SUBAPPLICATION CONSTRUCT_DDS_TOPIC (* Construct DDS Topic *)
  (* Standard: 61499-2 *)
  (* Version 1.0, 2023-03-15, Tim Hesse *)
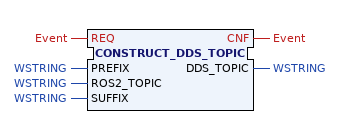
  EVENT_INPUT
    REQ; (* Normal Execution Request *)
  END_EVENT
  EVENT_OUTPUT
    CNF; (* Execution Confirmation *)
  END_EVENT
  VAR_INPUT
    PREFIX : WSTRING; (* Topic Prefix *)
    ROS2_TOPIC : WSTRING; (* ROS 2 Topic *)
    SUFFIX : WSTRING; (* Topic Suffix *)
  END_VAR
  VAR_OUTPUT
    DDS_TOPIC : WSTRING; (* DDS Topic *)
  END_VAR
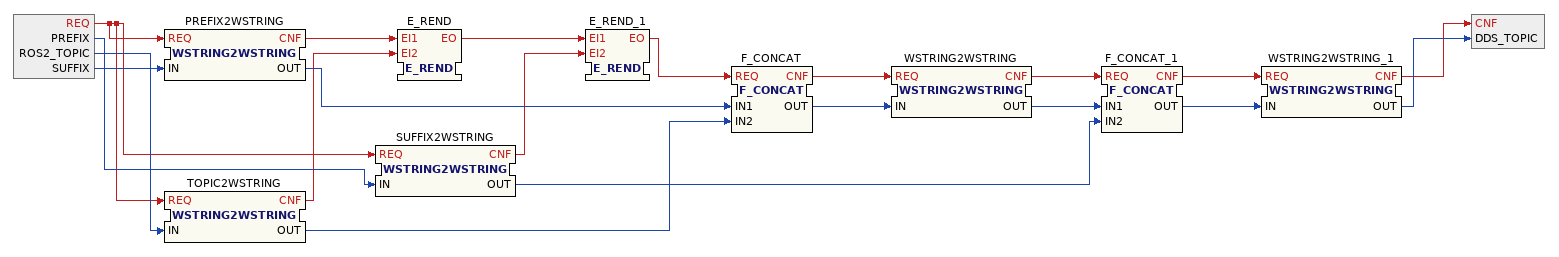
  FBS
    PREFIX2WSTRING : WSTRING2WSTRING;
    TOPIC2WSTRING : WSTRING2WSTRING;
    SUFFIX2WSTRING : WSTRING2WSTRING;
    E_REND : E_REND;
    E_REND_1 : E_REND;
    F_CONCAT : F_CONCAT;
    WSTRING2WSTRING : WSTRING2WSTRING;
    F_CONCAT_1 : F_CONCAT;
    WSTRING2WSTRING_1 : WSTRING2WSTRING;
  END_FBS
  EVENT_CONNECTIONS
    REQ TO PREFIX2WSTRING.REQ;
    REQ TO TOPIC2WSTRING.REQ;
    REQ TO SUFFIX2WSTRING.REQ;
    PREFIX2WSTRING.CNF TO E_REND.EI1;
    TOPIC2WSTRING.CNF TO E_REND.EI2;
    E_REND.EO TO E_REND_1.EI1;
    SUFFIX2WSTRING.CNF TO E_REND_1.EI2;
    F_CONCAT.CNF TO WSTRING2WSTRING.REQ;
    E_REND_1.EO TO F_CONCAT.REQ;
    WSTRING2WSTRING.CNF TO F_CONCAT_1.REQ;
    F_CONCAT_1.CNF TO WSTRING2WSTRING_1.REQ;
    WSTRING2WSTRING_1.CNF TO CNF;
  END_CONNECTIONS
  DATA_CONNECTIONS
    PREFIX TO PREFIX2WSTRING.IN;
    ROS2_TOPIC TO TOPIC2WSTRING.IN;
    SUFFIX TO SUFFIX2WSTRING.IN;
    PREFIX2WSTRING.OUT TO F_CONCAT.IN1;
    TOPIC2WSTRING.OUT TO F_CONCAT.IN2;
    F_CONCAT.OUT TO WSTRING2WSTRING.IN;
    WSTRING2WSTRING.OUT TO F_CONCAT_1.IN1;
    SUFFIX2WSTRING.OUT TO F_CONCAT_1.IN2;
    F_CONCAT_1.OUT TO WSTRING2WSTRING_1.IN;
    WSTRING2WSTRING_1.OUT TO DDS_TOPIC;
  END_CONNECTIONS
END_SUBAPPLICATION
